FUNCTION_BLOCK INTERNAL FINAL FB_ReadRepeatedFieldStringTests EXTENDS FB_TestSuite
VAR_INPUT
END_VAR
VAR_OUTPUT
END_VAR
VAR
    fbFieldCodecString : FB_FieldCodecString;
END_VAR

ShouldReadRepeatedFieldTheory();
ShouldReadNonConsecutiveRepeatedFields();

METHOD PRIVATE ShouldReadNonConsecutiveRepeatedFields
VAR CONSTANT
    (*
        message Demo {
            repeated uint32 a = 1;
            fixed32 b =2;
        }
        JSON:
        {
          "a": [
            0, 1, 2, 151
          ],
          "b": 321
        }
    *)
    cRawMessage : ARRAY[0..15] OF BYTE := [16#0A, 16#03, 16#00, 16#01, 16#02, 16#15, 16#41, 16#01, 16#00, 16#00, 16#0A, 16#02, 16#97, 16#01];
    cExpected   : ARRAY[0..15] OF BYTE := [0, 1, 2, 151];
END_VAR
VAR_INST
    stState : ST_ParserInternalState;
    fbFieldCodecInt32 : FB_FieldCodecInt32;
END_VAR
VAR
    aActual             : ARRAY [0..15] OF BYTE;
    hr                  : HRESULT;
    nActualFieldIndex   : UDINT;
    nTag                : UDINT;
    nB                  : UDINT;
END_VAR
TEST(__POUNAME());

// Arrange
stState.nBufferPos := 0;
stState.nBufferSize := SIZEOF(cRawMessage);

// Act
// Parses a=[0,1,2]: 16#0A, 16#03, 16#00, 16#01, 16#02
F_ParseTag(cRawMessage, stState, nTag=> );
hr := F_ReadRepeatedField(cRawMessage, stState, anyArray:= F_ToAnyType(aActual), anyFirstElem:= F_ToAnyType(aActual[0]), ipFieldCodec:= fbFieldCodecInt32, nFieldIndex:= nActualFieldIndex);

// Parses b=321: 16#15, 16#41, 16#01, 16#00, 16#00
F_ParseTag(cRawMessage, stState, nTag=> );
F_ParseRawLittleEndian32(cRawMessage, stState, nValue=> nB);

// Parses a=[151]: 16#0A, 16#02, 16#97, 16#01
F_ParseTag(cRawMessage, stState, nTag=> );
hr := F_ReadRepeatedField(cRawMessage, stState, anyArray:= F_ToAnyType(aActual), anyFirstElem:= F_ToAnyType(aActual[0]), ipFieldCodec:= fbFieldCodecInt32, nFieldIndex:= nActualFieldIndex);

// Assert
AssertEquals_DINT(
    Expected:= S_OK,
    Actual:= hr,
    Message:= 'Expected S_OK instead of error');
    
{warning disable C0041}
AssertArrayEquals_BYTE(Expecteds:= cExpected, Actuals:= aActual, Message:= '');
    
AssertEquals_UDINT(
    Expected:= 4,
    Actual:= nActualFieldIndex,
    Message:= CONCAT('Expected nActualFieldIndex to equal ', TO_STRING(4)));
    
TEST_FINISHED_NAMED(__POUNAME());
END_METHOD

METHOD PRIVATE ShouldReadRepeatedField
VAR_IN_OUT CONSTANT
    aBuffer     : ARRAY [*] OF BYTE;
    aExpected   : ARRAY [*] OF T_MAXSTRING;
END_VAR
VAR_INPUT CONSTANT
    nBufferPosStart     : UDINT;
    nExpectedBufferPos  : UDINT;
    nExpectedFieldIndex : UDINT;
    ipFieldCodec        : I_FieldCodec;
END_VAR
VAR_INST
    stState : ST_ParserInternalState;
END_VAR
VAR
    aActual             : ARRAY[0..15] OF T_MAXSTRING;
    hr                  : HRESULT;
    nActualFieldIndex   : UDINT;
    nTag                : UDINT;
    i                   : DINT;
END_VAR
// Arrange
stState.nBufferPos := nBufferPosStart;
stState.nBufferSize := TO_UDINT(UPPER_BOUND(aBuffer, 1) + 1);

// Act
F_ParseTag(aBuffer, stState, nTag=> nTag);
hr := F_ReadRepeatedField(aBuffer, stState, anyArray:= F_ToAnyType(aActual), anyFirstElem:= F_ToAnyType(aActual[0]), ipFieldCodec, nFieldIndex:= nActualFieldIndex);

// Assert
AssertEquals_DINT(
    Expected:= S_OK,
    Actual:= hr,
    Message:= 'Expected S_OK instead of error');
    
{warning disable C0041}
// AssertArrayEquals_(Expecteds:= aExpected, Actuals:= aActual, Message:= '');
FOR i := 0  TO UPPER_BOUND(aExpected, 1) DO 
    AssertEquals_STRING(Expected:= aExpected[i], Actual:= aActual[i], Message:= '');
END_FOR

AssertEquals_UDINT(
    Expected:= nExpectedBufferPos,
    Actual:= stState.nBufferPos,
    Message:= CONCAT('Expected stState.nBufferPos to equal ', TO_STRING(nExpectedBufferPos)));
    
AssertEquals_UDINT(
    Expected:= nExpectedFieldIndex,
    Actual:= nActualFieldIndex,
    Message:= CONCAT('Expected nActualFieldIndex to equal ', TO_STRING(nExpectedFieldIndex)));
END_METHOD

METHOD PRIVATE ShouldReadRepeatedFieldTheory : REFERENCE TO FB_Test
VAR CONSTANT
    cRawValueString1    : ARRAY[0..255] OF BYTE := [16#0A, 16#0B, 16#54, 16#65, 16#73, 16#74, 16#53, 16#74, 16#72, 16#69, 16#6E, 16#67, 16#30, 16#0A, 16#0B, 16#54, 16#65, 16#73, 16#74, 16#53, 16#74, 16#72, 16#69, 16#6E, 16#67, 16#31, 16#0A, 16#0B, 16#54, 16#65, 16#73, 16#74, 16#53, 16#74, 16#72, 16#69, 16#6E, 16#67, 16#32, 16#0A, 16#0B, 16#54, 16#65, 16#73, 16#74, 16#53, 16#74, 16#72, 16#69, 16#6E, 16#67, 16#33];
    
END_VAR

VAR CONSTANT
    aExpectedString1        : ARRAY[0..15] OF T_MAXSTRING := ['TestString0', 'TestString1', 'TestString2', 'TestString3'];
END_VAR

VAR
    viExpected : __SYSTEM.VAR_INFO;
    sAnyDummy   : T_MAXSTRING;
END_VAR
TEST(__POUNAME());

THIS^.fbFieldCodecString.SetAnyString(F_ToAnyString(sAnyDummy));
ShouldReadRepeatedField(aBuffer:= cRawValueString1, aExpected:= aExpectedString1, nBufferPosStart:= 0, nExpectedBufferPos:= 53, nExpectedFieldIndex:= 4, THIS^.fbFieldCodecString);

TEST_FINISHED_NAMED(__POUNAME());
END_METHOD

END_FUNCTION_BLOCK

(* stored: Version 1.1.0.1
   POU FB_ReadRepeatedFieldStringTests: Id {481fde89-a9de-4d33-b2f7-5458b704ebce}, SpecialFunc None
   Method ShouldReadNonConsecutiveRepeatedFields: Id {52cb7e82-bd02-4a86-a734-0d7e1470d8fb}
   Method ShouldReadRepeatedField: Id {ea7665fd-02f2-480a-9007-efe05cdec4ed}
   Method ShouldReadRepeatedFieldTheory: Id {e5fc16b6-2350-4421-bb6e-d4de18745678} *)
